VISUALIZATION VISU_State_red_green  // 12x17
VAR_IN_OUT
	state : BOOL;
END_VAR
    Ellipse (0,5 10x10), colour toggle: state
END_VISUALIZATION

(* stored: Version 1.1.0.1, ProductVersion 3.1.0.36
   Visu VISU_State_red_green: Id {d36d6dd2-b5ad-460b-acc3-72c9b418dd8e} *)
